FUNCTION_BLOCK BulkModulus
VAR_INPUT
END_VAR
VAR_OUTPUT
END_VAR
VAR
END_VAR

END_FUNCTION_BLOCK

(* stored: Version 1.1.0.1, ProductVersion 3.1.4024.9
   POU BulkModulus: Id {d896bbce-21be-40f0-ade7-5314da5b1d90}, SpecialFunc None *)
